{attribute 'qualified_only'}
VAR_GLOBAL
	GVL_MPG_Value : UINT;
END_VAR

(* stored: Version 1.1.0.1, ProductVersion 3.1.4024.11
   GVL Temp: Id {ba013bbf-fd0b-47c2-9325-6267efdb3ece} *)
